PROGRAM Doff_Angled
VAR
END_VAR

GVL.astAxes[AXIS_DOFF_ANGLED].stInputs.bLimitBwd := TRUE;
GVL.astAxes[AXIS_DOFF_ANGLED].stInputs.bLimitFwd := TRUE;
GVL.astAxes[AXIS_DOFF_ANGLED].stControl.bEnable := TRUE;

astAxes[AXIS_DOFF_ANGLED].stDescription.sAxisName := 'DOFF_ANGLED';

END_PROGRAM

(* stored: Version 1.1.0.1, ProductVersion 3.1.4024.12
   POU Doff_Angled: Id {963a6779-feb6-4643-bf35-ed9a0701229d}, SpecialFunc None *)
